// TIA Portal V16 export
// export: Created 2022-04-09T14:12:41.986226Z, ExportSetting WithDefaults, DisplayName Totally Integrated Automation Portal, DisplayVersion V16 Update 3, DisplayName TIA Portal Version Control Interface, DisplayVersion V16 Update 2, DisplayName TIA Portal Openness, DisplayVersion V16 Update 3, DisplayName STEP 7 Professional, DisplayVersion V16 Update 3, DisplayName STEP 7 Safety, DisplayVersion V16, DisplayName WinCC Professional, DisplayVersion V16 Update 3
FUNCTION "FC18151_StdSubTimeEventRTC" : Void   // FC18151, LAD
TITLE = Standard Module [SUBROUTINE] — Event Timer RTC
{ S7_Optimized_Access := 'TRUE' }
AUTHOR : M_Gledhill
FAMILY : Subroutine
NAME : StdSubTimeEventRTC
VERSION : 1.1
// PRACTICAL SERIES AUTOMATION LIBRARY (PAL)   —   COPYRIGHT 2020 – M. GLEDHILL (MIT LICENCE)
//                   ———— ◆ ————
// FULL ONLINE DOCUMENTATION IS AVAILABLE AT: https://practicalseries.com/2001-pal/index.html
// stored: AutoNumber false, IsIECCheckEnabled true, SetENOAutomatically false, UDAEnableTagReadback false
   VAR_INPUT
      TRIGGER : Bool;   // Trigger signal record start time on rising edge, end time on falling edge
   END_VAR
   VAR_IN_OUT
      DYNAMIC_DATA : "UT38151_Dy_SubTimeEventRTC";   // Dynamic data storage (UDT)
   END_VAR
   VAR_TEMP
      revInfo : "UT01000_St_SysRevision";   // Revision information for this block
      licInfo : "UT01001_St_SysLicence";   // Licence information for this block
      wrkInt : Int;   // Working storage area (integer)
      wrkReal : Real;   // Working storage area (real)
      wrkLInt : ULInt;   // Working storage area (long integer, unsigned)
   END_VAR
   VAR_TEMP   // added for the SCL form of the ladder/FBD networks
      _w1 : Bool;
      _w2 : Bool;
   END_VAR
BEGIN

REGION Network 1: Block description — Sections 1 to 3
   // ▄▄▄▄▄▄▄▄▄▄▄▄▄▄▄▄▄▄▄▄▄▄▄▄▄▄▄▄▄▄▄▄▄  ＳＴＡＮＤＡＲＤ  ▄▄ 
   // 
   // 
   // TITLE:    SUBROUTINE — EVENT TIMER RTC
   // 
   // 
   // ▀▀▀▀▀▀▀▀▀▀▀▀▀▀▀▀▀▀▀▀▀▀▀▀▀▀▀▀▀▀▀▀▀▀▀▀▀▀▀▀▀▀▀▀ 
   // 
   // ┌──────────────────────────────────────────┐
   // │                                          │
   // │          FC18151 — SOFTWARE MODULE DESIGN SPECIFICATION (SMDS)            │
   // │                                          │
   // │      The PDF version of the SMDS for this module is available online here:        │
   // │              http://psop.uk/pal-smds-fc18151-p              │
   // │                                          │
   // │      It is also available as part of the Project User Defined Documentation,      │
   // │      it can be accessed by selecting this module in the Project Tree          │
   // │      (on the left) and pressing SHIFT+F1                        │
   // │                                          │
   // └─────────────────────────────────────── ʷᴵᴰ⁻ᵇᵈʰ ┘
   // 
   // FC18151_SubTimeEventRTC is a subroutine block that times the duration of an event 
   // to nanosecond resolution.
   // 
   // The block records the time the event started (rising edge of the TRIGGER signal), the time the 
   // event ended (falling edge of the TRIGGER signal) and calculates the duration of the event (end 
   // time minus the start time).
   // 
   // The start and end times are read from the real time clock of the controller.
   // 
   // This is a subroutine block.
   // 
   // 
   // 
   // ▄▄▄▄▄▄▄▄▄▄▄▄▄▄▄▄▄▄▄▄▄▄▄▄▄▄▄▄▄▄▄▄▄▄▄▄▄▄▄▄▄▄▄▄
   // 1.     BLOCK TECHNICAL SUMMARY
   // 
   // 
   //  ――――――――――――――――――――――――――――――――――――――――――
   //  NOMENCLATURE & ADDRESSING
   //  ――――――――――――――――――――――――――――――――――――――――――
   //  BLOCK TITLE         Subroutine Event Timer using RTC
   //  BLOCK FUNCTION GROUP    Subroutine
   //  BLOCK ADDRESS       FC18151
   //  BLOCK SYMBOL        FC18151_SubTimeEventRTC
   //  BLOCK USER ID         SubTimeEventRTC
   // 
   //  ――――――――――――――――――――――――――――――――――――――――――
   //  BLOCK TYPE & USAGE
   //  ――――――――――――――――――――――――――――――――――――――――――
   //  BLOCK TYPE         Function (FC)
   //  BLOCK NUMBER        18151
   //  LANGUAGE           LAD
   //  OPTIMISED ACCESS     Yes
   //  PAL USAGE TYPE       Standard block
   // 
   //  ――――――――――――――――――――――――――――――――――――――――――
   //  METRICS
   //  ――――――――――――――――――――――――――――――――――――――――――
   //  EXECUTION TIME       18.4 μs¹
   //  LOAD MEMORY       21.4 kB
   //  WORK MEMORY           0.4 kB  
   //  ――――――――――――――――――――――――――――――――――――――――――
   //                ¹ Measured on: CPU-1515-2PN (order no. 6ES7512-2AM02-0AB0) 
   //                             http://psop.uk/pal-ds-cpu1515
   // 
   // 
   // 
   // ▂▂▂▂▂▂▂▂▂▂▂▂▂▂▂▂▂▂▂▂▂▂▂▂▂▂▂▂▂▂▂▂▂▂▂▂▂▂▂▂▂▂▂▂
   // 1.1      Additional document references
   // 
   // 
   // Only those documents specified in OB1 (section DOCUMENT REFERENCES) are listed within this 
   // block. There are no additional document references.
   // 
   //                ━━━   ⬙⬙⬙⬙⬙⬙   ━━━
   // 
   // 
   // 
   // ▄▄▄▄▄▄▄▄▄▄▄▄▄▄▄▄▄▄▄▄▄▄▄▄▄▄▄▄▄▄▄▄▄▄▄▄▄▄▄▄▄▄▄▄
   // 2.     FUNCTIONAL DESCRIPTION
   // 
   // 
   // FC18151 is the Subroutine Event Timer using RTC block, it simply records the duration of an event 
   // with a high degree of accuracy. The event being timed is a Boolean signal passed to the block as 
   // the TRIGGER parameter.
   // 
   // Three times are recorded for the event, the start time (rising edge of the TRIGGER parameter), the 
   // end time (falling edge of the TRIGGER parameter) and the duration of the event (end time minus 
   // the start time). The duration is calculated on the falling edge of the TRIGGER parameter, 
   // immediately after the end time is recorded.
   // 
   // The start and end times are read from the Controller’s internal real time clock (RTC) and are 
   // stored in DTL (date time long) format, this format contains year, month, day, hours, minutes, 
   // seconds, milliseconds, microseconds and nano seconds.
   // 
   // The duration is stored in LTime (long time, 64-bit) format, and is very accurate, it resolves to 
   // days, hours, minutes, seconds milliseconds, microseconds and nanoseconds, it keeps this 
   // resolution irrespective of the duration.
   // 
   // The duration is also calculated as a real number in seconds (or fractions thereof); this is a 
   // more convenient format for holding the duration, but is not as accurate as the LTime format.
   // 
   // 
   // 
   // ▄▄▄▄▄▄▄▄▄▄▄▄▄▄▄▄▄▄▄▄▄▄▄▄▄▄▄▄▄▄▄▄▄▄▄▄▄▄▄▄▄▄▄▄
   // 3.     DETAILED BLOCK DESCRIPTION
   // 
   // The purpose of this block is to determine with a high degree of accuracy the duration of an event, 
   // the event itself must be in the form of a Boolean trigger signal, the rising edge of the signal is 
   // considered to be the start of the event and the falling edge the end of the event.
   // 
   // The event signal is passed to the block as the TRIGGER parameter. 
   // The block returns five values, these are stored in a UDT passed to the block in the 
   // DYNAMIC_DATA parameter: 
   // 
   //  ――――――――――――――――――――――――――――――――――――――――――
   //  PARAM         ASSOCIATED UDT            ASSOCIATED DATA BLOCK
   //  ――――――――――――――――――――――――――――――――――――――――――
   //  DYNAMIC_DATA     UT38151_Dy_SubTimeEventRTC       DB38151_Dy_SubTimeEventRTC
   //  ――――――――――――――――――――――――――――――――――――――――――
   // 
   // 
   // The block returns the following data:
   // 
   //  UT38151_Dy_SubTimeEventRTC
   //  ―――――――――――――――――――――――――――――――――――――――――― 
   //  SIGNAL NAME          FUNCTION                     TYPE
   //  ――――――――――――――――――――――――――――――――――――――――――
   //  status_Running      STATUS — The event timer is running         Bool
   // 
   //  actual_StartTime      ACTUAL — Time at which the TRIGGER signal        DTL
   //                      went high (event start time)
   // 
   //  actual_EndTime        ACTUAL — Time at which the TRIGGER signal     DTL
   //                      went low (event end time)
   // 
   //  actual_Duration        ACTUAL — Event duration              LTime
   // 
   //  actual_DurationSec       ACTUAL — Event duration in seconds           REAL
   //  ――――――――――――――――――――――――――――――――――――――――――
   // 
   // 
   // 
   // ▂▂▂▂▂▂▂▂▂▂▂▂▂▂▂▂▂▂▂▂▂▂▂▂▂▂▂▂▂▂▂▂▂▂▂▂▂▂▂▂▂▂▂▂
   // 3.1     Timing an event
   // 
   // The block constantly monitors the TRIGGER parameter; if a rising edge is seen on the TRIGGER 
   // parameter (point ① in the figure below), the Controller RTC is read and its value is stored in 
   // actual_StartTime, at the same time the running signal (status_Running) is activated.
   // 
   // The block continues to monitor the TRIGGER parameter, when a falling edge is detected 
   // (point ②), the RTC is read once more and its value is stored in actual_EndTime, and the running 
   // signal (status_Running) is deactivated.
   // 
   // Once the end time is stored, the following calculation is carried out:
   // 
   // 
   // ┌───────────────────────────┐
   // │ actual_Duration =  actual_EndTime ─ actual_StartTime    │
   // └───────────────────────────┘
   // 
   // 
   //                     ①            ②
   //   TRIGGER │             ┏━━━━━━━━━━━━┓
   //         │             ┃               ┃
   //         │             ┃               ┃
   //         │             ┃               ┃
   //         │             ┃               ┃                              
   //         ┼━━━━━━━━━━━━╶╶╶╶╶╶╶╶╶╶╶╶╶━━━━━━━━━━ time
   //                  ↗             ↖
   //          actual_Start_Time ╎            ╎ actual_End_Time
   //    DTL#2020-04-18-09:34:25.899548353        DTL#2020-04-18-09:34:36.004744916
   // 
   //                    ╎               ╎                      actual_Duration
   //                                      LT#10S_105MS_196US_563NS
   //                    ╎               ╎  
   //                                                     actual_DurationSec
   //                    ╎               ╎                              10.10519
   // 
   //         │status_Running      ┏━━━━━━━━━━━━┓
   //         │             ┃               ┃
   //         │             ┃               ┃
   //         │             ┃               ┃
   //         │             ┃               ┃
   //         ┼━━━━━━━━━━━━╶╶╶╶╶╶╶╶╶╶╶╶╶━━━━━━━━━━
   // 
   // 
   // 
   // ▂▂▂▂▂▂▂▂▂▂▂▂▂▂▂▂▂▂▂▂▂▂▂▂▂▂▂▂▂▂▂▂▂▂▂▂▂▂▂▂▂▂▂▂
   // 3.1     Date and time data types
   // 
   // Both the start and end times (actual_StartTime and actual_EndTime) are of the type DTL 
   // (date time long), this itself is a data structure in the form:
   // 
   //  DTL Data Structure
   //  ――――――――――――――――――――――――――――――――――――――――――
   //  SIGNAL NAME          FUNCTION                     TYPE
   //  ――――――――――――――――――――――――――――――――――――――――――
   //  YEAR             Year (returns a value in the range 1970 to 2262)     UInt
   //  MONTH            Month (1-12 representing Jan to Dec)        USInt
   //  DAY              Day of month (1-31)                USInt
   //  WEEKDAY          Day of week (1-7, where 1=Sunday, 7=Saturday)    USInt
   //  HOUR           Hour of day (0-23)                   USInt
   //  MINUTE           Minutes (0-59)                   USInt
   //  SECOND            Seconds (0-59)                  USInt
   //  NANOSECOND        Nanoseconds (0-999,999,999)           UDint
   //  ――――――――――――――――――――――――――――――――――――――――――
   // 
   // When displayed, it has the format:
   // 
   //       DTL#2020-04-18-09:34:25.899548353
   // 
   //  I.e.      18th April 2020 at 09:43:25 AM and 899,548,353 ns.
   // 
   // The calculated duration (actual_Duration) is of data type LTime (long time).
   // 
   // The LTime data type is essentially an 8-byte number (64-bit number) that stores a time value in 
   // nanoseconds. In the above example, the actual_Duration has the formatted value of:
   // 
   //       LT#10S_105MS_196US_563NS
   // 
   //  I.e.      10 seconds, 105 milliseconds, 196 microseconds and 563 nanoseconds.
   // 
   // It is shown in this format, because TIA portal understands the LTime data type and is able to 
   // interpret the value as days, hours, minute, seconds, milliseconds, microseconds and 
   // nanoseconds. 
   // 
   // In practice, the actual_Duration simply (in this example) holds a very large number:
   // 
   //       10,105,196,563
   // 
   // This is the duration of the event in nanoseconds (i.e. 10,105,196,563 nanoseconds). To convert 
   // the number to seconds, simply divide by 1,000,000,000 (or 1 × 10^9); this would give:
   // 
   //       10.105196563 seconds
   // 
   // The reason the duration is specified as an LTime rather that DTL is that, somewhat confusingly, 
   // DTL is a relative measure of time (relative to 1st January, 1970), if the above duration were 
   // represented as a DTL value it would read:
   // 
   //       DTL#1970-01-01-00:00:10.105196563
   // 
   // Hours, minutes and seconds are OK, but the date part doesn’t make sense (to make it 
   // meaningful, 1970 must be subtracted from the YEAR value and 1 from both the MONTH and 
   // DAY values).
   // 
   // The LTime data type can store a duration of up to 106,751 days (about 300 years) and while not 
   // perfect, it seems long enough for most practical situations (possibly not for geological 
   // applications).
   // 
   // The actual_Duration in LTime format is very accurate, but it is an unwieldly data type, to provide a 
   // more user friendly (although less accurate) format, the actual_Duration signal is converted to a 
   // real number giving the duration in seconds, this is stored in the actual_DurationSec signal. In the 
   // above example: 
   // 
   //       actual_DurationSec has the value 10.10519 seconds
   // 
   // It is less accurate, it does not resolve to nanoseconds; however, it is easier to use and display 
   // and is accurate enough for most applications.
   // 
   // 
   // 
   // ▁▁▁▁▁▁▁▁▁▁▁▁▁▁▁▁▁▁▁▁▁▁▁▁▁▁▁▁▁▁▁▁▁▁▁▁▁▁▁▁▁▁▁▁
   // A note on real numbers (and accuracy)
   // 
   // The LTime format is very accurate, it is basically counting nanoseconds, and because it is 64-bits 
   // long it can count up to very high values (about 292 years at nanosecond resolution).
   // 
   // Real numbers however, are limited to 32-bits and suffer from precision loss, this results from the 
   // fact that the real number has an accuracy of “about” 7 decimal digits, for example 20365.45, 
   // 20.43728, 1.482967, 0.3356428, &c. Essentially, the bigger the number, the fewer the decimal 
   // places — a total of 7 decimal digits.
   // 
   // Very big and very small numbers can be represented by adding trailing zeros for big numbers 
   // (e.g. 3275625000) and leading zeros for small numbers (0.000003275625) in both these 
   // examples, there are only 7 decimal digits, just shifted effectively left or right.
   // 
   // This type of representation is usually handled by applying scientific notation, the number 
   // 1,568,497,000,000 would be represented as 1.568497 × 10^12, it only has 7 decimal digits, 
   // the number 1,568,497,132,792, would be represented as exactly the same value, the 132,792 
   // part of the number can not be resolved and are lost.
   // 
   //                ━━━   ⬙⬙⬙⬙⬙⬙   ━━━
   // 
   // 
   // 
   // ▄▄▄▄▄▄▄▄▄▄▄▄▄▄▄▄▄▄▄▄▄▄▄▄▄▄▄▄▄▄▄▄▄▄▄▄▄▄▄▄▄▄▄▄
   // 4.     Supervisory system interface
   // 
   // 
   // FC18151 is a Subroutine block. It does not have a supervisory system interface.
   // 
   // 
   //                ━━━   ⬙⬙⬙⬙⬙⬙   ━━━
   // 
   // 
   // 
   // ▄▄▄▄▄▄▄▄▄▄▄▄▄▄▄▄▄▄▄▄▄▄▄▄▄▄▄▄▄▄▄▄▄▄▄▄▄▄▄▄▄▄▄▄
   // 5.     PARAMETERS
   // 
   // 
   // The following parameters are associated with the block:
   // 
   //  
   //  ――――――――――――――――――――――――――――――――――――――――――
   //  PARAM         FUNCTION                    TYPE      IN-OUT 
   //  ――――――――――――――――――――――――――――――――――――――――――
   //  TRIGGER       Event trigger signal (a rising edge marks the     Bool   In
   //           start of the event, the falling edge the end)
   // 
   // 
   //  DYNAMIC_DATA      Stores the results of the event timing       UT38151    InOut
   //  ――――――――――――――――――――――――――――――――――――――――――
   // 
   // Note:    FC18151 is one of the few blocks that does not require the SYS_SIGNALS parameter 
   //      (this has been done to make minimise the block interface)
   // 
   //                ━━━   ⬙⬙⬙⬙⬙⬙   ━━━
   // 
   // 
   // 
   // ▄▄▄▄▄▄▄▄▄▄▄▄▄▄▄▄▄▄▄▄▄▄▄▄▄▄▄▄▄▄▄▄▄▄▄▄▄▄▄▄▄▄▄▄
   // 6.     DATA STRUCTURES AND USAGE
   // 
   // 
   // The block has the following associated data structure:
   // 
   // 
   //  ――――――――――――――――――――――――――――――――――――――――――
   //  DATA STRUCTURE             DESCRIPTION
   //  ――――――――――――――――――――――――――――――――――――――――――
   //  UT01000_St_SysRevision          Revision information for this block    See FC01001
   //  UT01001_St_SysLicence           Licence information for this block  See FC01001
   //  UT38151_Dy_SubTimeEventRTC        Dynamic data structure for the event timing block
   //  ――――――――――――――――――――――――――――――――――――――――――
   // 
   // 
   // 
   // ▂▂▂▂▂▂▂▂▂▂▂▂▂▂▂▂▂▂▂▂▂▂▂▂▂▂▂▂▂▂▂▂▂▂▂▂▂▂▂▂▂▂▂▂
   // 6.1     UT38151_Dy_TimeEventRTC
   // 
   // Stores the timing values for the event:
   // 
   //  UT38151_Dy_TimeEventRTC
   //  ――――――――――――――――――――――――――――――――――――――――――
   //  SIGNAL NAME          FUNCTION                     TYPE
   //  ――――――――――――――――――――――――――――――――――――――――――
   //  status_Running      STATUS — The event timer is running         Bool
   // 
   //  actual_StartTime      ACTUAL — Time at which the TRIGGER signal        DTL
   //                      went high (event start time)
   // 
   //  actual_EndTime        ACTUAL — Time at which the TRIGGER signal     DTL
   //                      went low (event end time)
   // 
   //  actual_Duration        ACTUAL — Event duration              LTime
   // 
   //  actual_DurationSec       ACTUAL — Event duration in seconds           REAL
   //  ――――――――――――――――――――――――――――――――――――――――――
   // 
   //                ━━━   ⬙⬙⬙⬙⬙⬙   ━━━
   // 
   // 
   // 
   // ▄▄▄▄▄▄▄▄▄▄▄▄▄▄▄▄▄▄▄▄▄▄▄▄▄▄▄▄▄▄▄▄▄▄▄▄▄▄▄▄▄▄▄▄
   // 7.     CONSTANTS AND TEMPORARY (LOCAL) DATA
   // 
   // 
   // 
   // ▂▂▂▂▂▂▂▂▂▂▂▂▂▂▂▂▂▂▂▂▂▂▂▂▂▂▂▂▂▂▂▂▂▂▂▂▂▂▂▂▂▂▂▂
   // 7.1     Constants
   // 
   // 
   // No constants are used in this block.
   // 
   // 
   // 
   // ▂▂▂▂▂▂▂▂▂▂▂▂▂▂▂▂▂▂▂▂▂▂▂▂▂▂▂▂▂▂▂▂▂▂▂▂▂▂▂▂▂▂▂▂
   // 7.2     Temporary (local) data
   // 
   // 
   // The following temporary data is used:
   // 
   //  ――――――――――――――――――――――――――――――――――――――――――
   //  SIGNAL NAME          FUNCTION                  TYPE
   //  ――――――――――――――――――――――――――――――――――――――――――
   //  revInfo             Revision information for the block         UT01000
   //  licInfo           Licensing information for the block      UT01001
   //  wrkInt           Working storage area (integer)          Int
   //  wrkReal           Working storage (Real)             Real
   //  wrkLInt            Working storage area (longinteger)      LInt
   //  ――――――――――――――――――――――――――――――――――――――――――
   // 
   //                ━━━   ⬙⬙⬙⬙⬙⬙   ━━━
   // 
   // 
   // 
   // ▄▄▄▄▄▄▄▄▄▄▄▄▄▄▄▄▄▄▄▄▄▄▄▄▄▄▄▄▄▄▄▄▄▄▄▄▄▄▄▄▄▄▄▄
   // 8.     BLOCK CALLS AND ASSOCIATIONS
   // 
   // 
   // This section details any blocks which may be called from within this software module (subroutine 
   // functions for example), any partner blocks with which it may be associated (for example a 
   // receive module that is partner with a transmit module &c.). It lists any system functions which 
   // may be called (e.g. reading the real time clock) and any system data types that may be used.
   // 
   // Finally, it lists any special calling requirements for the block (for example, must be called from 
   // within a cyclic interrupt organisation block) and if the block is using “optimised access” (this is 
   // the default arrangement).
   // 
   // 
   // 
   // ▂▂▂▂▂▂▂▂▂▂▂▂▂▂▂▂▂▂▂▂▂▂▂▂▂▂▂▂▂▂▂▂▂▂▂▂▂▂▂▂▂▂▂▂
   // 8.1     Block calls from within this module
   // 
   // 
   // There are no PAL block calls from within this block.
   // 
   // 
   // 
   // ▂▂▂▂▂▂▂▂▂▂▂▂▂▂▂▂▂▂▂▂▂▂▂▂▂▂▂▂▂▂▂▂▂▂▂▂▂▂▂▂▂▂▂▂
   // 8.2     Blocks associated with this module
   // 
   // 
   // This is a stand-alone block and is not associated with any other blocks.
   // 
   // 
   // 
   // ▂▂▂▂▂▂▂▂▂▂▂▂▂▂▂▂▂▂▂▂▂▂▂▂▂▂▂▂▂▂▂▂▂▂▂▂▂▂▂▂▂▂▂▂
   // 8.3     System block calls and system data typesThe following calls are made to system blocks:
   // 
   // 
   //  System block calls
   //  ――――――――――――――――――――――――――――――――――――――――――
   //  BLOCK          TITLE             DESCRIPTION  
   //  ――――――――――――――――――――――――――――――――――――――――――
   //  RD_LOC_T             Read the local RTC time    Reads the CPU real time clock 
   //  ――――――――――――――――――――――――――――――――――――――――――
   // 
   // There are no special system data types used.
   // 
   // 
   // 
   // ▂▂▂▂▂▂▂▂▂▂▂▂▂▂▂▂▂▂▂▂▂▂▂▂▂▂▂▂▂▂▂▂▂▂▂▂▂▂▂▂▂▂▂▂
   // 8.4     Special properties and requirements
   // 
   // 
   // 
   // ▁▁▁▁▁▁▁▁▁▁▁▁▁▁▁▁▁▁▁▁▁▁▁▁▁▁▁▁▁▁▁▁▁▁▁▁▁▁▁▁▁▁▁▁
   // 8.4.1     Block optimisation, IEC compatibility and library conformance
   // 
   // 
   //    •   Block optimisation is ACTIVE for this block.
   // 
   //    •   The block has been checked for IEC compatibility and is compliant.
   // 
   //    •   The block is compatible with all IEC library-conformance module constraints
   // 
   // 
   // 
   // ▁▁▁▁▁▁▁▁▁▁▁▁▁▁▁▁▁▁▁▁▁▁▁▁▁▁▁▁▁▁▁▁▁▁▁▁▁▁▁▁▁▁▁▁
   // 8.4.2     Calling requirements
   // 
   // 
   // There are no special calling requirements for this block.
   // 
   //                ━━━   ⬙⬙⬙⬙⬙⬙   ━━━
   // 
   // 
   // 
   // ▄▄▄▄▄▄▄▄▄▄▄▄▄▄▄▄▄▄▄▄▄▄▄▄▄▄▄▄▄▄▄▄▄▄▄▄▄▄▄▄▄▄▄▄
   // 9.     EXAMPLE USAGE
   // 
   // 
   // The following shows a typical deployment of FC18151:
   // 
   //                      ┌─────────────
   //        ──────────────┤ FC18151
   //                      ├───────────
   //                 %M100.0    │
   //               "Event001"   ─┤ TRIGGER
   //                      │
   //     "DB38151_Dy_TimeEventRTC".Event001 ─┤ DYNAMIC_DATA
   //                      │
   //                      │             │
   //                                    │
   //                           ─────────┘
   // 
   //               ━━━   ⬙⬙⬙⬙⬙⬙   ━━━
   // 
   // 
   // 
   // ▄▄▄▄▄▄▄▄▄▄▄▄▄▄▄▄▄▄▄▄▄▄▄▄▄▄▄▄▄▄▄▄▄▄▄▄▄▄▄▄▄▄▄▄
   // 10.     TEST AND VERIFICATION PATH
   // 
   // 
   // The following diagram shows the full test and verification path for the formal release of each 
   // version of the software module. See the Test Plan [Ref. 003] for full details, available here:
   //         http://psop.uk/pal-tp-p
   // 
   // 
   //         FC18151-T001         FC18151-T002
   // 
   //     Test version: 000.801     Test version: 001.801
   //  Released version: 001.000     Released version: 002.000
   // Released commit: D0003    Released commit: D0011
   // 
   //        SCR      SMT              SCV     
   // ＿＿＿＿＿＿┌┐＿＿ ▛▜ ＿＿＿＿＿＿＿＿＿＿＿＿╓╖＿＿
   //       └┘   ▙▟             ╙╜  
   // Initial test           Comments standardised
   // 
   // Initial test to release the      Comments updated & 
   // module following the      minor typographical 
   // development stage.       corrections
   // Full SMT              SCV only
   // 
   // 
   // Where:
   // ――――――――――――――――――――――――――――――――――――――――――――
   //  SCR    Source Code Review      A visual inspection of the software to ensure it has been written  
   // ┌┐             to the correct standards, uses the correct structures within the
   // └┘             software and is generally suitable for deployment.               
   // 
   //  SMT Software Module Test    A full and detailed test of an individual software module in
   //   ▛▜              isolation; such testing requires that all branches of the 
   //   ▙▟              software are tested. 
   // 
   //                It tests all the interfaces to the module, any data recorded or 
   //                stored by the module, all error and exception handling functions 
   //                and tests all timed and interrupt driven operations.
   // 
   //  SCV Software Compatibility     A mechanism for verifying that no executable code software 
   // ╓╖    Verification          changes have been made to a module following changes to
   // ╙╜             comment fields.
   // 
   //                Allows typographical errors &c. to be corrected without forcing 
   //                a full SMT on a module that has not functionally changed.
   // ――――――――――――――――――――――――――――――――――――――――――――
   // 
   // An SCV can only be performed on a module that has at some point previously, successfully 
   // completed both an SCR and SMT. Where an SCV is implemented, it replaces the requirement for 
   // both the SCR and the SMT for the test iteration in question.
   // 
   //                ━━━   ⬙⬙⬙⬙⬙⬙   ━━━
   // 
   // 
   // 
   // ██████████████ █ █ █ █  END   █ █ █ █ ██████████████
END_REGION

REGION Network 2: Current revision and modification history
   // ▄▄▄▄▄▄▄▄▄▄▄▄▄▄▄▄▄▄▄▄▄▄▄▄▄▄▄▄▄▄▄▄▄▄▄▄▄▄▄▄▄▄▄▄
   // MODIFICATION HISTORY
   // 
   // 
   // The revision data shown here, in the network comments, contains additional information 
   // reflecting the software development workflow under the version control system (VCS) employed 
   // to track all software changes.
   // 
   // The VCS in use is the Git Source Code Management system in conjunction with the GitHub online 
   // hosting system. The software in its entirety is available in the GitHub remote repository:
   // 
   //      https://github.com/practicalseries/PS2001-pal-software
   // 
   // The repository is public and can be freely copied (forked in GitHub terminology) and used 
   // under the MIT licence. 
   // 
   // The MIT licence is reproduced in full in the last network of this software module
   // 
   // 
   //  ―――――――――――――――――――――――――――――――――――――――――――
   //  DATE       REVISION             MASTER BRANCH     DEV
   //          (nnn.amm)   COMMIT TAG    (Base ---> Merge)    BRANCH   Author
   //  ———————————————————————————————————————————
   //  2022.04.08    001.101   D0010A-000.104   D0010 N/A     D010A   M. Gledhill
   //                        Comments updated and standardised
   //                        NW 2 comments combined with NW 1
   // 
   //  2021.02.19    001.000   D0003      D0002 D0003  None    M. Gledhill
   //                        FC18151 — RELEASED FOR USE
   //                          Merge back to master branch
   // 
   //  2021.02.19    001.000   D0002A-001.000   D0002 N/A     D0002A   M. Gledhill
   //                        FC18151 — Post test RELEASED FOR USE
   //  
   //  2021.02.18    000.801   D0002A-000.801   D0002 N/A     D0002A   M. Gledhill
   //                        FC18151 Migration to VCS — Released for test
   //  ———————————————————————————————————————————
   //   Where: nnn  =  Major revision
   //         a  =  Type (1-7 Development, 8 Proving, 9 Qualification, 0 Release)
   //       mm  =  Minor revision (must be 00 if a = 0)
   //         Block properties version number should be set to nn.a (only one decimal place)
   // 
   // ▄▄▄▄▄▄▄▄▄▄▄▄▄▄▄▄▄▄▄▄▄▄▄▄▄▄▄▄▄▄▄▄▄▄▄▄▄▄▄▄▄▄▄▄
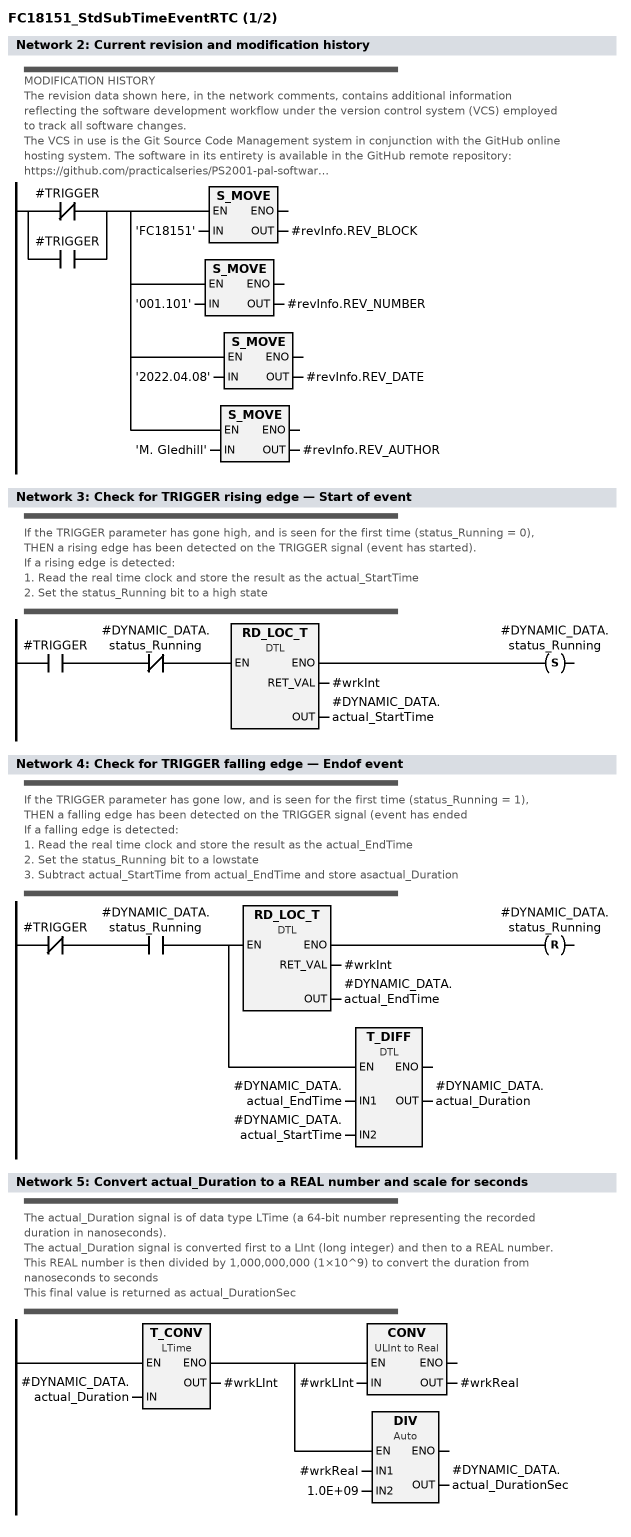
   RUNG wire#powerrail
      I_Contact( #TRIGGER )
      wire#w1
      S_Move(in := 'FC18151', out => #revInfo.REV_BLOCK)
   END_RUNG
   RUNG wire#powerrail
      Contact( #TRIGGER )
   END_RUNG wire#w1
   RUNG wire#w1
      S_Move(in := '001.101', out => #revInfo.REV_NUMBER)
   END_RUNG
   RUNG wire#w1
      S_Move(in := '2022.04.08', out => #revInfo.REV_DATE)
   END_RUNG
   RUNG wire#w1
      S_Move(in := 'M. Gledhill', out => #revInfo.REV_AUTHOR)
   END_RUNG
   // the same network as SCL:
   IF NOT #TRIGGER OR #TRIGGER THEN
       #revInfo.REV_BLOCK := 'FC18151';
       #revInfo.REV_NUMBER := '001.101';
       #revInfo.REV_DATE := '2022.04.08';
       #revInfo.REV_AUTHOR := 'M. Gledhill';
   END_IF;
END_REGION

REGION Network 3: Check for TRIGGER rising edge — Start of event
   // ▀▀▀▀▀▀▀▀▀▀▀▀▀▀▀▀▀▀▀▀▀▀▀▀▀▀▀▀▀▀▀▀▀▀▀▀▀▀▀▀▀▀▀▀
   // If the TRIGGER parameter has gone high, and is seen for the first time (status_Running = 0),
   // THEN a rising edge has been detected on the TRIGGER signal (event has started).
   // 
   // If a rising edge is detected:
   //   1. Read the real time clock and store the result as the actual_StartTime
   //   2. Set the status_Running bit to a high state
   // ▄▄▄▄▄▄▄▄▄▄▄▄▄▄▄▄▄▄▄▄▄▄▄▄▄▄▄▄▄▄▄▄▄▄▄▄▄▄▄▄▄▄▄▄
   RUNG wire#powerrail
      Contact( #TRIGGER )
      I_Contact( #DYNAMIC_DATA.status_Running )
      { S7_Templates := "date_type := DTL" } RD_LOC_T(RET_VAL => #wrkInt, OUT => #DYNAMIC_DATA.actual_StartTime)
      S_Coil( #DYNAMIC_DATA.status_Running )
   END_RUNG
   // the same network as SCL:
   #wrkInt := RD_LOC_T(EN := #TRIGGER AND NOT #DYNAMIC_DATA.status_Running,
                       OUT => #DYNAMIC_DATA.actual_StartTime,
                       ENO => #_w1);
   IF #_w1 THEN #DYNAMIC_DATA.status_Running := TRUE; END_IF;
END_REGION

REGION Network 4: Check for TRIGGER falling edge — Endof event
   // ▀▀▀▀▀▀▀▀▀▀▀▀▀▀▀▀▀▀▀▀▀▀▀▀▀▀▀▀▀▀▀▀▀▀▀▀▀▀▀▀▀▀▀▀
   // If the TRIGGER parameter has gone low, and is seen for the first time (status_Running = 1),
   // THEN a falling edge has been detected on the TRIGGER signal (event has ended
   // 
   // If a falling edge is detected:
   //   1. Read the real time clock and store the result as the actual_EndTime
   //   2. Set the status_Running bit to a lowstate
   //   3. Subtract actual_StartTime from actual_EndTime and store asactual_Duration
   // ▄▄▄▄▄▄▄▄▄▄▄▄▄▄▄▄▄▄▄▄▄▄▄▄▄▄▄▄▄▄▄▄▄▄▄▄▄▄▄▄▄▄▄▄
   RUNG wire#powerrail
      I_Contact( #TRIGGER )
      Contact( #DYNAMIC_DATA.status_Running )
      wire#w1
      { S7_Templates := "date_type := DTL" } RD_LOC_T(RET_VAL => #wrkInt, OUT => #DYNAMIC_DATA.actual_EndTime)
      R_Coil( #DYNAMIC_DATA.status_Running )
   END_RUNG
   RUNG wire#w1
      { S7_Templates := "[date_type := DTL, time_type := LTime]" } T_DIFF(IN1 := #DYNAMIC_DATA.actual_EndTime, IN2 := #DYNAMIC_DATA.actual_StartTime, OUT => #DYNAMIC_DATA.actual_Duration)
   END_RUNG
   // the same network as SCL:
   #wrkInt := RD_LOC_T(EN := NOT #TRIGGER AND #DYNAMIC_DATA.status_Running,
                       OUT => #DYNAMIC_DATA.actual_EndTime,
                       ENO => #_w1);
   #_w2 := NOT #TRIGGER AND #DYNAMIC_DATA.status_Running;
   IF #_w1 THEN #DYNAMIC_DATA.status_Running := FALSE; END_IF;
   IF #_w2 THEN
       T_DIFF(IN1 := #DYNAMIC_DATA.actual_EndTime,
              IN2 := #DYNAMIC_DATA.actual_StartTime,
              OUT => #DYNAMIC_DATA.actual_Duration);
   END_IF;
END_REGION

REGION Network 5: Convert actual_Duration to a REAL number and scale for seconds
   // ▀▀▀▀▀▀▀▀▀▀▀▀▀▀▀▀▀▀▀▀▀▀▀▀▀▀▀▀▀▀▀▀▀▀▀▀▀▀▀▀▀▀▀▀
   // The actual_Duration signal is of data type LTime (a 64-bit number representing the recorded
   // duration in nanoseconds).
   // 
   // The actual_Duration signal is converted first to a LInt (long integer) and then to a REAL number.
   // 
   // This REAL number is then divided by 1,000,000,000 (1×10^9) to convert the duration from 
   // nanoseconds to seconds
   // 
   // This final value is returned as actual_DurationSec
   // ▄▄▄▄▄▄▄▄▄▄▄▄▄▄▄▄▄▄▄▄▄▄▄▄▄▄▄▄▄▄▄▄▄▄▄▄▄▄▄▄▄▄▄▄
   RUNG wire#powerrail
      { S7_Templates := "[src_type := LTime, dest_type := ULInt]" } T_CONV(IN := #DYNAMIC_DATA.actual_Duration, OUT => #wrkLInt)
      wire#w1
      { S7_Templates := "[SrcType := ULInt, DestType := Real]" } Convert(in := #wrkLInt, out => #wrkReal)
   END_RUNG
   RUNG wire#w1
      Div(in1 := #wrkReal, in2 := 1.0E+09, out => #DYNAMIC_DATA.actual_DurationSec)
   END_RUNG
   // the same network as SCL:
   T_CONV(IN := #DYNAMIC_DATA.actual_Duration, OUT => #wrkLInt, ENO => #_w1);
   IF #_w1 THEN
       #wrkReal := ULINT_TO_REAL(#wrkLInt);
       #DYNAMIC_DATA.actual_DurationSec := #wrkReal / 1.0E+09;
   END_IF;
END_REGION

REGION Network 6: LICENCE AND CONTACT INFORMATION
   // ▀▀▀▀▀▀▀▀▀▀▀▀▀▀▀▀▀▀▀▀▀▀▀▀▀▀▀▀▀▀▀▀▀▀▀▀▀▀▀▀▀▀▀▀
   // LICENCE AND CONTACT INFORMATION
   // 
   // This software and its associated documentation is made available under the MIT Licence:
   // 
   // ════════════════════════════════════════════
   // 
   // The MIT License (MIT)
   // 
   // Copyright © 2020 Michael Gledhill
   // 
   // Permission is hereby granted, free of charge, to any person obtaining a copy of this software 
   // and associated documentation files (the “Software”), to deal in the Software without restriction, 
   // including without limitation the rights to use, copy, modify, merge, publish, distribute, 
   // sublicense, and/or sell copies of the Software, and to permit persons to whom the Software is 
   // furnished to do so, subject to the following conditions: 
   // 
   // The above copyright notice and this permission notice shall be included in all copies or 
   // substantial portions of the Software.
   // 
   // THE SOFTWARE IS PROVIDED “AS IS”, WITHOUT WARRANTY OF ANY KIND, EXPRESS OR IMPLIED, 
   // INCLUDING BUT NOT LIMITED TO THE WARRANTIES OF MERCHANTABILITY, FITNESS FOR A 
   // PARTICULAR PURPOSE AND NON-INFRINGEMENT. IN NO EVENT SHALL THE AUTHORS OR COPYRIGHT 
   // HOLDERS BE LIABLE FOR ANY CLAIM, DAMAGES OR OTHER LIABILITY, WHETHER IN AN ACTION OF 
   // CONTRACT, TORT OR OTHERWISE, ARISING FROM, OUT OF OR IN CONNECTION WITH THE SOFTWARE 
   // OR THE USE OR OTHER DEALINGS IN THE SOFTWARE.
   // 
   // ════════════════════════════════════════════
   //                    ┌────────────┐
   // You can reach the author by email here:   │  mg@practicalseries.com  │
   //                    └────────────┘
   // Questions, corrections, constructive criticism and complaints (polite ones) are invited.
   // 
   // ▄▄▄▄▄▄▄▄▄▄▄▄▄▄▄▄▄▄▄▄▄▄▄▄▄▄▄▄▄▄▄▄▄▄▄▄▄▄▄▄▄▄▄▄
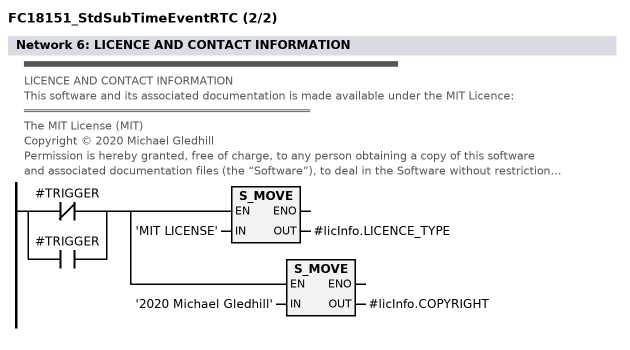
   RUNG wire#powerrail
      I_Contact( #TRIGGER )
      wire#w1
      S_Move(in := 'MIT LICENSE', out => #licInfo.LICENCE_TYPE)
   END_RUNG
   RUNG wire#powerrail
      Contact( #TRIGGER )
   END_RUNG wire#w1
   RUNG wire#w1
      S_Move(in := '2020 Michael Gledhill', out => #licInfo.COPYRIGHT)
   END_RUNG
   // the same network as SCL:
   IF NOT #TRIGGER OR #TRIGGER THEN
       #licInfo.LICENCE_TYPE := 'MIT LICENSE';
       #licInfo.COPYRIGHT := '2020 Michael Gledhill';
   END_IF;
END_REGION
END_FUNCTION
